PROGRAM IoT
VAR CONSTANT
	EC_MASTER_NETID : T_AmsNetId := '192.168.80.1.4.1';
END_VAR
VAR
	sdo_controller : FB_CoeSdoAccess(sNetId := EC_MASTER_NETID);
	planar_tiles_diag_data: ARRAY[1..2] OF sdo_xplanar_aps_diag;
	sessions: ARRAY [1..2] OF CoeSdoCommand;
	read_cycle_timer: TON;
	fbMqttPublish : FB_mqtt_publish;
END_VAR



// Get diganosis data from SDO
sdo_controller();
fbMqttPublish();

// Get diagnostics data every 0.5s
read_cycle_timer(IN := NOT read_cycle_timer.Q, PT := T#500MS);

IF read_cycle_timer.Q THEN
	sdo_controller.query(
					nSlaveAddr := 1001,
					bCompleteAccess := TRUE, 
					nIndex := 16#FA00, 
					nSubIndex := 0,
					pDstBuf := ADR(planar_tiles_diag_data[1]),
					cbBufLen := SIZEOF(planar_tiles_diag_data[1]),
					event_handler := fbMqttPublish
					);
	sdo_controller.query(
					nSlaveAddr := 1003,
					bCompleteAccess := TRUE, 
					nIndex := 16#FA00, 
					nSubIndex := 0,
					pDstBuf := ADR(planar_tiles_diag_data[2]),
					cbBufLen := SIZEOF(planar_tiles_diag_data[2]),
					event_handler := fbMqttPublish
					);
END_IF

END_PROGRAM

(* stored: Version 1.1.0.1, ProductVersion 3.1.4024.12
   POU IoT: Id {a18040ea-08a5-44c3-a275-8f9a987457b9}, SpecialFunc None *)
